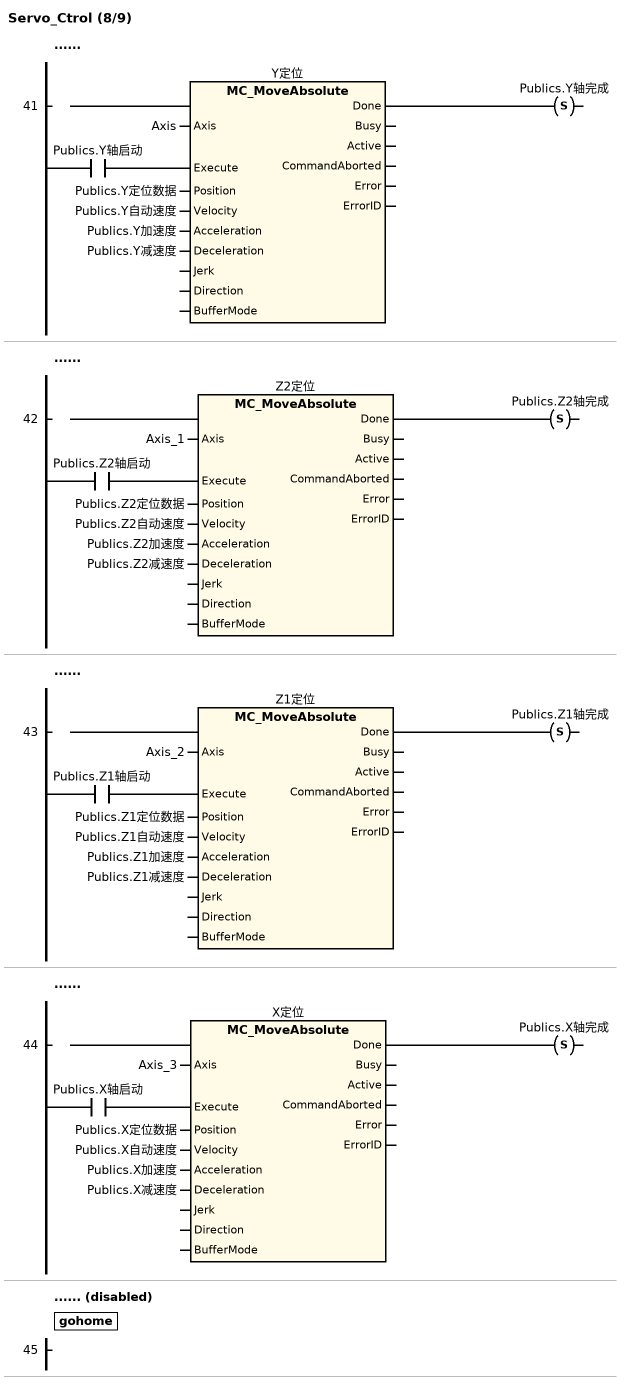
// NETWORK 41: ......
Y定位(
    Axis := Axis,
    Execute := Publics.Y轴启动,
    Position := Publics.Y定位数据,
    Velocity := Publics.Y自动速度,
    Acceleration := Publics.Y加速度,
    Deceleration := Publics.Y减速度); // MC_MoveAbsolute
Publics.Y轴完成 S= Y定位.Done;

// NETWORK 42: ......
Z2定位(
    Axis := Axis_1,
    Execute := Publics.Z2轴启动,
    Position := Publics.Z2定位数据,
    Velocity := Publics.Z2自动速度,
    Acceleration := Publics.Z2加速度,
    Deceleration := Publics.Z2减速度); // MC_MoveAbsolute
Publics.Z2轴完成 S= Z2定位.Done;

// NETWORK 43: ......
Z1定位(
    Axis := Axis_2,
    Execute := Publics.Z1轴启动,
    Position := Publics.Z1定位数据,
    Velocity := Publics.Z1自动速度,
    Acceleration := Publics.Z1加速度,
    Deceleration := Publics.Z1减速度); // MC_MoveAbsolute
Publics.Z1轴完成 S= Z1定位.Done;

// NETWORK 44: ......
X定位(
    Axis := Axis_3,
    Execute := Publics.X轴启动,
    Position := Publics.X定位数据,
    Velocity := Publics.X自动速度,
    Acceleration := Publics.X加速度,
    Deceleration := Publics.X减速度); // MC_MoveAbsolute
Publics.X轴完成 S= X定位.Done;

// NETWORK 45: ...... (disabled)
// label: gohome

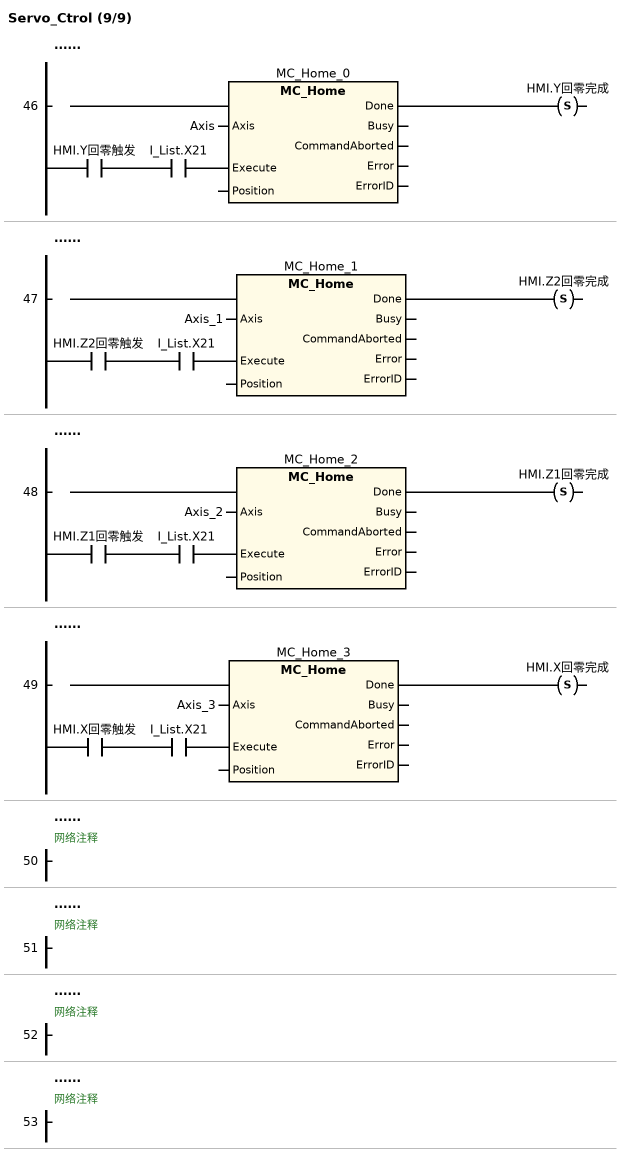
// NETWORK 46: ......
MC_Home_0(Axis := Axis, Execute := HMI.Y回零触发 AND I_List.X21); // MC_Home
HMI.Y回零完成 S= MC_Home_0.Done;

// NETWORK 47: ......
MC_Home_1(Axis := Axis_1, Execute := HMI.Z2回零触发 AND I_List.X21); // MC_Home
HMI.Z2回零完成 S= MC_Home_1.Done;

// NETWORK 48: ......
MC_Home_2(Axis := Axis_2, Execute := HMI.Z1回零触发 AND I_List.X21); // MC_Home
HMI.Z1回零完成 S= MC_Home_2.Done;

// NETWORK 49: ......
MC_Home_3(Axis := Axis_3, Execute := HMI.X回零触发 AND I_List.X21); // MC_Home
HMI.X回零完成 S= MC_Home_3.Done;

// NETWORK 50: ......
// 网络注释

// NETWORK 51: ......
// 网络注释

// NETWORK 52: ......
// 网络注释

// NETWORK 53: ......
// 网络注释

END_PROGRAM

// Device/Application/POU
PROGRAM POU
VAR
	当前步: uint;
	下一步: uint;
	定位位置: ARRAY[0..3] OF Lreal;
	LS_4AxisLine_0: LS_4AxisLine;
	避开扫描周期: BOOL;
	所有轴启动: BOOL;
	轴运行完成: BOOL;
END_VAR
VAR // added by the converter: edge detectors and wires of the graphical bodies
    _w1, _w2, _w3, _w4, _w5, _w6, _w7, _w8, _w9, _w10, _w11, _w12 : BOOL;
END_VAR

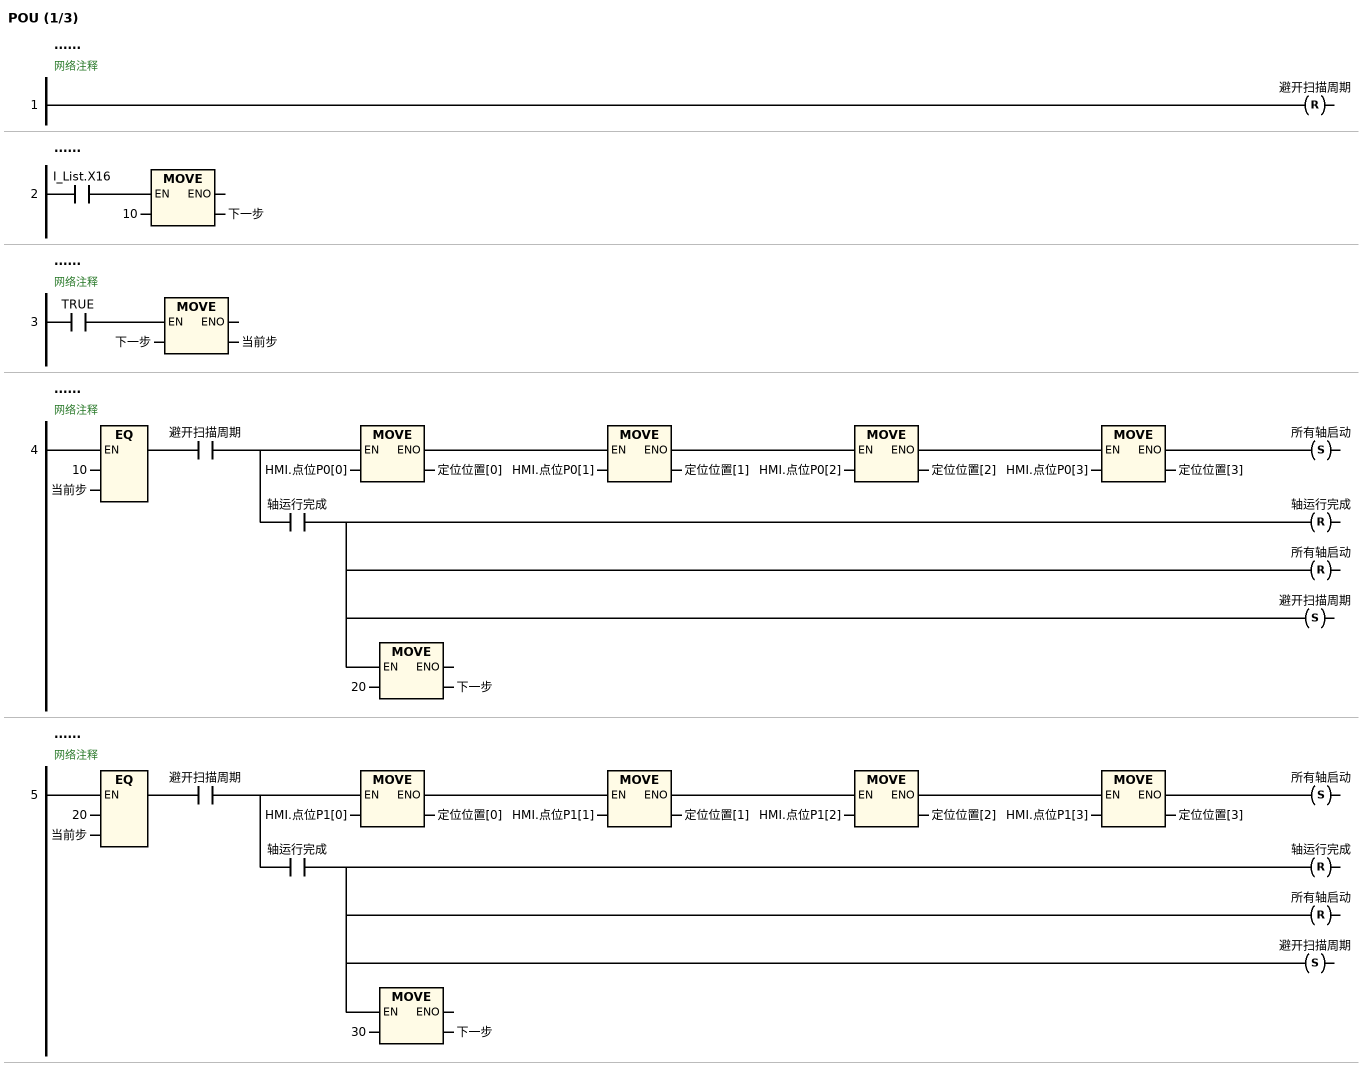
// NETWORK 1: ......
// 网络注释
避开扫描周期 R= TRUE;

// NETWORK 2: ......
IF I_List.X16 THEN 下一步 := 10; END_IF

// NETWORK 3: ......
// 网络注释
当前步 := 下一步;

// NETWORK 4: ......
// 网络注释
_w1 := 10 = 当前步 AND 避开扫描周期;
IF _w1 THEN 定位位置[0] := HMI.点位P0[0]; END_IF
IF _w1 THEN 定位位置[1] := HMI.点位P0[1]; END_IF
IF _w1 THEN 定位位置[2] := HMI.点位P0[2]; END_IF
IF _w1 THEN 定位位置[3] := HMI.点位P0[3]; END_IF
所有轴启动 S= _w1;
_w2 := _w1 AND 轴运行完成;
轴运行完成 R= _w2;
所有轴启动 R= _w2;
避开扫描周期 S= _w2;
IF _w2 THEN 下一步 := 20; END_IF

// NETWORK 5: ......
// 网络注释
_w3 := 20 = 当前步 AND 避开扫描周期;
IF _w3 THEN 定位位置[0] := HMI.点位P1[0]; END_IF
IF _w3 THEN 定位位置[1] := HMI.点位P1[1]; END_IF
IF _w3 THEN 定位位置[2] := HMI.点位P1[2]; END_IF
IF _w3 THEN 定位位置[3] := HMI.点位P1[3]; END_IF
所有轴启动 S= _w3;
_w4 := _w3 AND 轴运行完成;
轴运行完成 R= _w4;
所有轴启动 R= _w4;
避开扫描周期 S= _w4;
IF _w4 THEN 下一步 := 30; END_IF

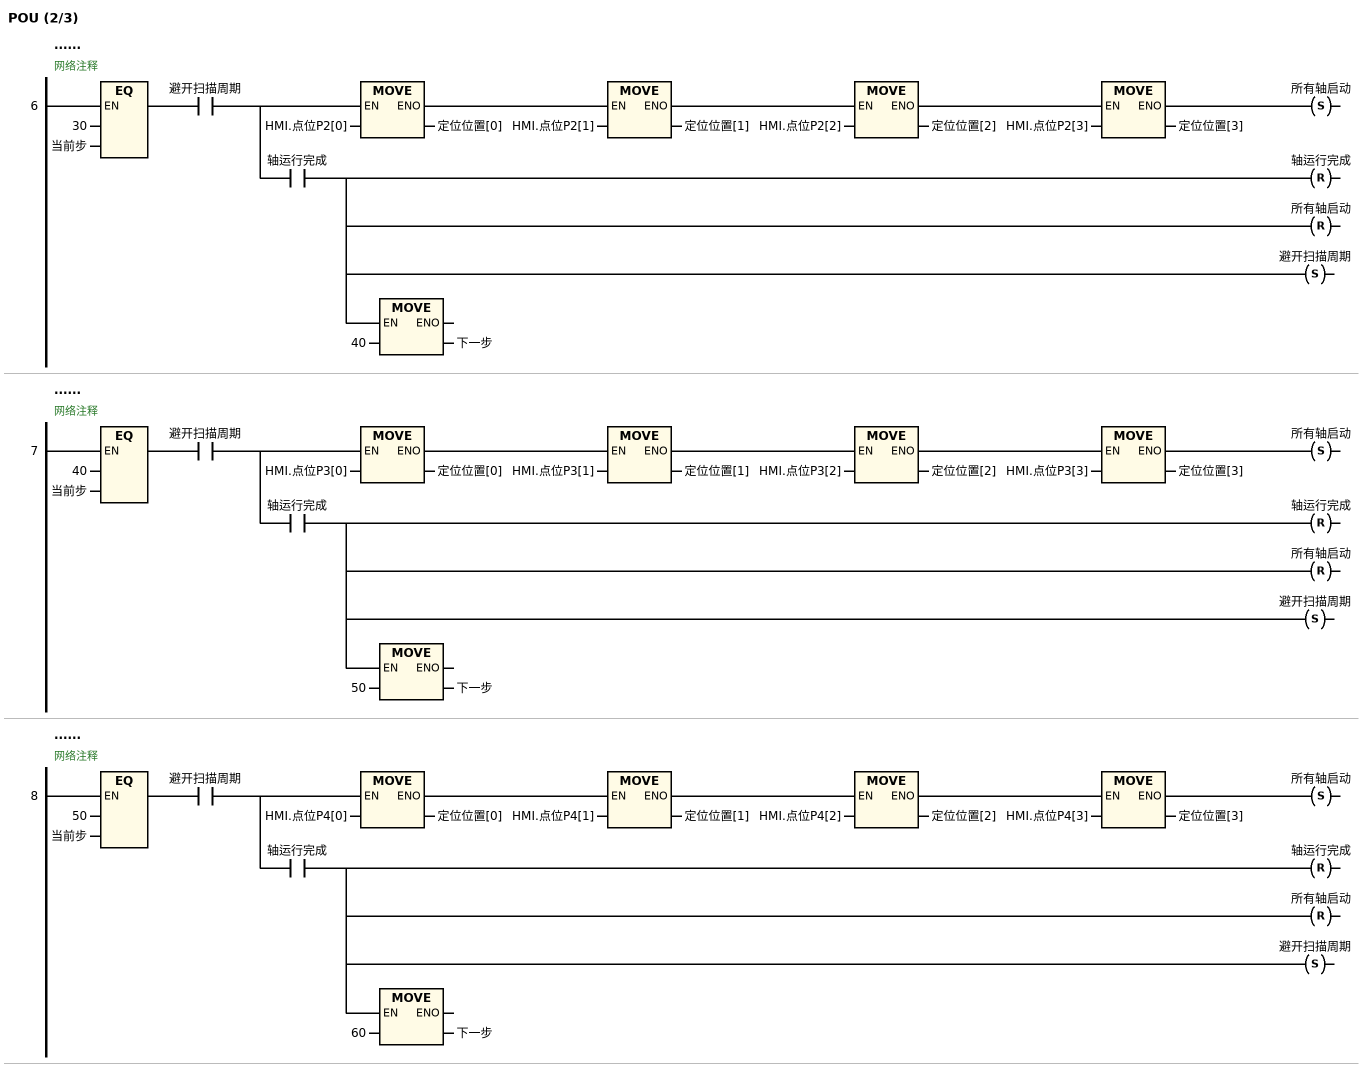
// NETWORK 6: ......
// 网络注释
_w5 := 30 = 当前步 AND 避开扫描周期;
IF _w5 THEN 定位位置[0] := HMI.点位P2[0]; END_IF
IF _w5 THEN 定位位置[1] := HMI.点位P2[1]; END_IF
IF _w5 THEN 定位位置[2] := HMI.点位P2[2]; END_IF
IF _w5 THEN 定位位置[3] := HMI.点位P2[3]; END_IF
所有轴启动 S= _w5;
_w6 := _w5 AND 轴运行完成;
轴运行完成 R= _w6;
所有轴启动 R= _w6;
避开扫描周期 S= _w6;
IF _w6 THEN 下一步 := 40; END_IF

// NETWORK 7: ......
// 网络注释
_w7 := 40 = 当前步 AND 避开扫描周期;
IF _w7 THEN 定位位置[0] := HMI.点位P3[0]; END_IF
IF _w7 THEN 定位位置[1] := HMI.点位P3[1]; END_IF
IF _w7 THEN 定位位置[2] := HMI.点位P3[2]; END_IF
IF _w7 THEN 定位位置[3] := HMI.点位P3[3]; END_IF
所有轴启动 S= _w7;
_w8 := _w7 AND 轴运行完成;
轴运行完成 R= _w8;
所有轴启动 R= _w8;
避开扫描周期 S= _w8;
IF _w8 THEN 下一步 := 50; END_IF

// NETWORK 8: ......
// 网络注释
_w9 := 50 = 当前步 AND 避开扫描周期;
IF _w9 THEN 定位位置[0] := HMI.点位P4[0]; END_IF
IF _w9 THEN 定位位置[1] := HMI.点位P4[1]; END_IF
IF _w9 THEN 定位位置[2] := HMI.点位P4[2]; END_IF
IF _w9 THEN 定位位置[3] := HMI.点位P4[3]; END_IF
所有轴启动 S= _w9;
_w10 := _w9 AND 轴运行完成;
轴运行完成 R= _w10;
所有轴启动 R= _w10;
避开扫描周期 S= _w10;
IF _w10 THEN 下一步 := 60; END_IF

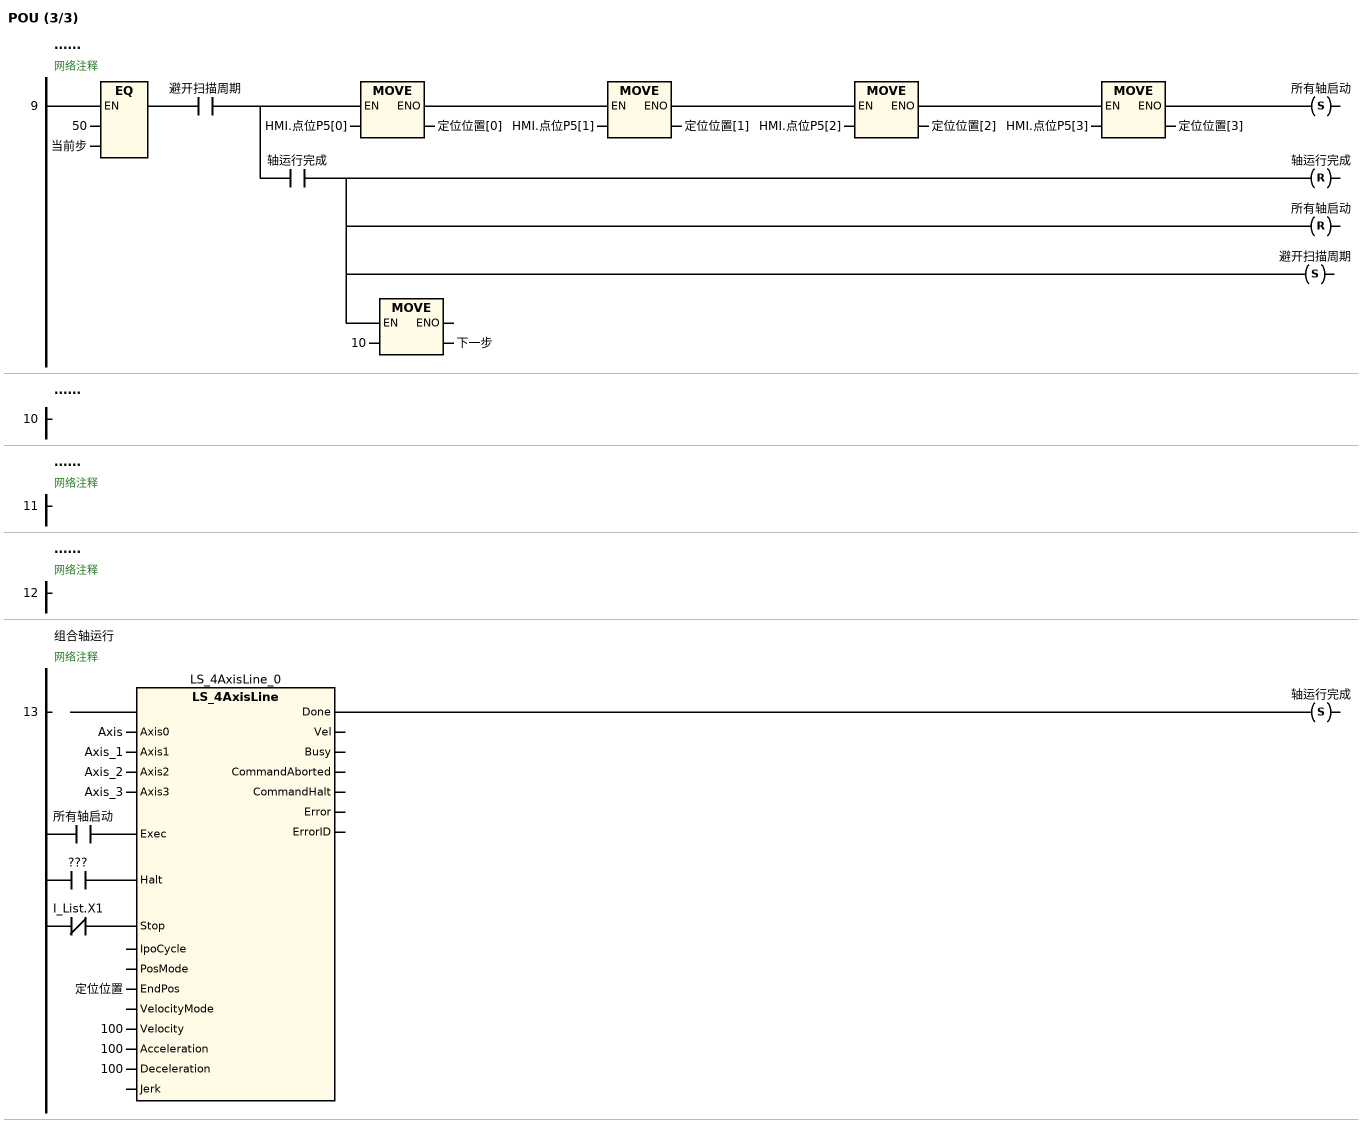
// NETWORK 9: ......
// 网络注释
_w11 := 50 = 当前步 AND 避开扫描周期;
IF _w11 THEN 定位位置[0] := HMI.点位P5[0]; END_IF
IF _w11 THEN 定位位置[1] := HMI.点位P5[1]; END_IF
IF _w11 THEN 定位位置[2] := HMI.点位P5[2]; END_IF
IF _w11 THEN 定位位置[3] := HMI.点位P5[3]; END_IF
所有轴启动 S= _w11;
_w12 := _w11 AND 轴运行完成;
轴运行完成 R= _w12;
所有轴启动 R= _w12;
避开扫描周期 S= _w12;
IF _w12 THEN 下一步 := 10; END_IF

// NETWORK 10: ......

// NETWORK 11: ......
// 网络注释

// NETWORK 12: ......
// 网络注释

// NETWORK 13: 组合轴运行
// 网络注释
LS_4AxisLine_0(
    Axis0 := Axis,
    Axis1 := Axis_1,
    Axis2 := Axis_2,
    Axis3 := Axis_3,
    Exec := 所有轴启动,
    Stop := NOT I_List.X1,
    EndPos := 定位位置,
    Velocity := 100,
    Acceleration := 100,
    Deceleration := 100); // LS_4AxisLine
轴运行完成 S= LS_4AxisLine_0.Done;

END_PROGRAM

// Device/Application/ITF
INTERFACE ITF

END_INTERFACE

// Device/Application/FunctionBlock/FB_CylinderDouble
FUNCTION_BLOCK FB_CylinderDouble
VAR_IN_OUT
	///气缸控制、状态和报警
	stCylvar: CYLINDER_REF;
END_VAR
VAR_INPUT
	///安全条件
	xReady: BOOL;
	///报警复位
	xReset: BOOL;
	///手动控制,每on一次,则反转输出点状态
	xManuCmd: BOOL;
	///原位检测
	xBackSensor: BOOL;
	///到位检测
	xFrontSensor: BOOL;
	///手自动不一致报警无效
	xManuAlmDisable: BOOL;
	///原位检测无效
	xBackSensorDisable: BOOL;
	///到位检测无效	
	xFrontSensorDisable: BOOL;
	///原位延时	
	wBackDelay: WORD;
	///到位延时
	wFrontDelay: WORD;
END_VAR
VAR_OUTPUT
	///输出点,对应双控气缸原位电磁阀
	xOutputA: BOOL;
	///输出点,应双控气缸到位电磁阀
	xOutputB: BOOL;
	///未满足安全条件报警
	f_xNotRdyAlm: BOOL;
	///手自动不一致报警	
	f_xManuAlm: BOOL;
	///未在原位报警
	f_xBackAlm: BOOL;
	///未到位报警	
	f_xFrontAlm: BOOL;
	///气缸处于不受控制状态报警
	f_xUncontrolledAlm: BOOL;
END_VAR
VAR
	///获取自动控制的上升沿
	fbAutoRise: R_TRIG;
	///获取自动控制的下升沿
	fbAutoFall: F_TRIG;
	///获取手动控制的下升沿
	fbManuFall: F_TRIG;
	///获取复位信号的上升沿
	fbResetRise: R_TRIG;
	///原位状态延时,用于输出原位状态
	fbBackTon: TON;
	///到位状态延时,用于输出到位状态	
	fbFrontTon: TON;
	///获取原位状态下降沿
	fbBackFall: F_TRIG;
	///获取到位状态下降沿
	fbFrontFall: F_TRIG;
	///原位动作超时,用于输出未在原位位置报警
	fbBackWait: TON;
	///到位动作超时,用于输出未在原位位置报警
	fbFrontWait: TON;
END_VAR

   //初始化时返回原位
   IF  xReady AND stCylvar.xInit AND ( NOT xManuCmd ) THEN
	     xOutputA  := TRUE; 
         xOutputB  := FALSE;
		 f_xManuAlm  := FALSE;
		 stCylvar.xInit  := FALSE;	  	  	 	  
   END_IF	  
   
   //获取手动控制、自动控制的边沿信号
   fbManuFall(CLK:=xManuCmd , Q=> );
   fbAutoRise(CLK:=stCylvar.xAutoCmd , Q=> );
   fbAutoFall(CLK:=stCylvar.xAutoCmd , Q=> );
   
   //1,手动操作时，如果满足安全条件且未屏蔽手自动不一致报警时，则输出点A反转，输出点B取输出点A的反逻辑
   IF xReady AND (NOT xManuAlmDisable) AND fbManuFall.Q THEN
	   xOutputA  := NOT xOutputA; 
	   xOutputB  := NOT xOutputA;
	   
	//手动操作生效时，判断输出点状态与自动命令是否一致，不一致时,置位手动操作执行中报警；一致时复位该报警。
	//当因安全条件不满足导致自动命令未执行时，可通过手动操作控制其动作执行,此时手动操作并不引起手动操作执行中报警。
   	   IF (stCylvar.xAutoCmd AND (NOT xManuAlmDisable) ) XOR xOutputB THEN
   	   	    f_xManuAlm  :=TRUE;
   	   ELSE 
   	   	    f_xManuAlm  :=FALSE;
   	   END_IF
   END_IF
   //2,手动操作时，如果满足安全条件且屏蔽了手自动不一致报警时，则自动控制点反转、复位手自动不一致报警，  
    IF xReady AND  xManuAlmDisable AND fbManuFall.Q THEN
   	    stCylvar.xAutoCmd  := NOT stCylvar.xAutoCmd ;
		f_xManuAlm  :=FALSE;		  	 	
    END_IF
   
   //自动命令置位时，如满足安全条件，则输出点A复位、 输出点B置位。
   IF xReady AND fbAutoRise.Q THEN
   	    xOutputA  :=FALSE;
		xOutputB  :=TRUE;
		
   END_IF
   //自动命令复位时，如满足安全条件，则输出点A置位、 输出点B复位。
   IF xReady AND fbAutoFall.Q THEN
   	    xOutputA  :=TRUE;
		xOutputB  :=FALSE;		
   END_IF
   
   
   //到位状态输出
   fbFrontTon(IN:=( NOT xOutputA ) AND xOutputB AND ( xFrontSensor OR xFrontSensorDisable ) AND ( NOT xBackSensor ) , PT:= WORD_TO_TIME ( wFrontDelay *10 ), Q=> stCylvar.xIsFront, ET=> );
   
   //原位状态输出
   fbBackTon(IN:= xOutputA  AND ( NOT xOutputB) AND ( NOT xFrontSensor ) AND ( xBackSensor OR xBackSensorDisable ) , PT:= WORD_TO_TIME ( wBackDelay *10 ) , Q=> stCylvar.xIsBack, ET=> );
   
   
   //报警复位
   fbResetRise(CLK:= xReset, Q=> );
   IF fbResetRise.Q THEN
   	   f_xNotRdyAlm := FALSE;
	   f_xFrontAlm := FALSE;
	   f_xBackAlm := FALSE;
	   f_xUncontrolledAlm := FALSE;
   
   END_IF
   
   
   //未满足安全条件报警
   //当手动操作或自动命令状态发生改变时，如果不能满足安全条件，则输出未满足安全条件报警
   IF ( fbManuFall.Q OR fbAutoRise.Q OR fbAutoFall.Q ) AND ( NOT xReady ) THEN
   	   f_xNotRdyAlm := TRUE; 
   END_IF
   
   
   //未在原位报警
   //自动命令变OFF后(上电后气缸处于自由状态时不判断)，延时5秒，如果原位标志未变为ON、且未发生手动操作和安全条件报警，则输出未到原位报警
   fbBackWait(IN:= ( NOT stCylvar.xAutoCmd ) AND ( xOutputA OR xOutputB ) , PT:= T#5S , Q=> , ET=> );
   fbBackFall(CLK:= stCylvar.xIsBack , Q=> );
   IF (( fbBackWait.Q AND (NOT stCylvar.xIsBack )) OR (( NOT stCylvar.xAutoCmd ) AND fbBackFall.Q )) AND  ( NOT f_xManuAlm ) AND  ( NOT f_xNotRdyAlm ) THEN
   	    f_xBackAlm := TRUE;
   END_IF
   
   
   //未在到位报警
   //自动命令变ON后，延时5秒，如果到位标志未变为ON、且未发生手动操作和安全条件报警，则输出未到位报警
   fbFrontWait(IN:= stCylvar.xAutoCmd , PT:= T#5S , Q=> , ET=> );
   fbFrontFall(CLK:= stCylvar.xIsFront, Q=> );
   IF ( ( fbFrontWait.Q AND ( NOT stCylvar.xIsFront ) ) OR (stCylvar.xAutoCmd AND fbFrontFall.Q )) AND ( NOT f_xManuAlm ) AND ( NOT f_xNotRdyAlm ) THEN
   	    f_xFrontAlm := TRUE;   
   END_IF      
   
   
   //不受控状态报警
   IF NOT ( xOutputA OR xOutputB ) THEN
   	    f_xUncontrolledAlm := TRUE;
   END_IF

END_FUNCTION_BLOCK
